(* CODESYS project ExampleRandomNumber.project

Project tree, tasks and I/O mapping:
  Device : CODESYS Control Win V3, 3S - Smart Software Solutions GmbH, order no. 305021, version 3.5.5.20
    application Application
      libraries: Standard, * (System)
      task MainTask (cyclic, interval t#20ms, priority 1) calls PLC_PRG_LD, PLC_PRG
      program PLC_PRG [ST]
      function rand [ST]
      global variables GVL
      program PLC_PRG_LD [LD]
  Rand/
    function rand [ST]
    program TestRand [ST]
*)

// Device/Application/GVL
VAR_GLOBAL
	randNext : ULINT := 42; //required external variable with a seed
END_VAR

// Device/Application/PLC_PRG_LD
//Test rand(), random number generator
PROGRAM PLC_PRG_LD
VAR
	number : UINT;
END_VAR

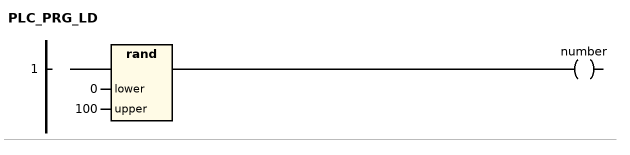
// NETWORK 1
number := rand(lower := 0, upper := 100);

END_PROGRAM

// Rand/rand
///Exempel: Generera slumptal mellan 1 ooch 10. 
///randNext : ULINT := 42;
///x : uint := rand(1,10)
///Ger ett slumptal mellan lower och upper
///Kräver att man har definierat en variabel randNext:ULINT:=<ett frö>;
///Ref: Bilting, U. Vägen Till C. Studentlitteratur. 2011.
FUNCTION rand : UINT
VAR_INPUT
	lower: UINT;
	upper: UINT;
END_VAR
VAR
	range: UINT := ((upper - lower) + 1);
	interval: UINT := (c4 / range);
	preRand: UINT;
END_VAR
VAR CONSTANT
	c1: UDINT := 1103515245;
	c2: UINT := 12345;
	c3: UDINT := 65536;
	c4: UINT := 32768;
END_VAR

randNext := randNext * c1 + c2;
preRand := ULINT_TO_UINT((randNext/c3) MOD c4);
IF interval > 0 THEN
	rand := (preRand+lower*interval-1)/interval; 
ELSE
	rand := preRand;
END_IF;
RETURN;

END_FUNCTION

// Device/Application/rand
//Example: Generate random numbers 1..10. 
//randNext : ULINT := 42; //required external variable with a seed
//x : uint := rand(1,10)
//
//Brief: Will give you a random number between lower och upper
//Requires an external variable: randNext:ULINT:=<seed>;
//Ref: Bilting, U. Vägen Till C. Studentlitteratur. 2011.
//
// Created by: Alexander Jaworowski 2015-02-05
// github.com/alexjaw/randomGenerator
FUNCTION rand : UINT
VAR_INPUT
	lower:UINT;
	upper:UINT;
END_VAR
VAR
	range:UINT:=upper-lower+1;
	interval:UINT:=c4/range;
	preRand:UINT;
END_VAR
VAR CONSTANT
	c1:UDINT:=1103515245;
	c2:UINT:=12345;
	c3:UDINT:=65536;
	c4:UINT:=32768;
END_VAR

randNext := randNext * c1 + c2;
preRand := ULINT_TO_UINT((randNext/c3) MOD c4);
IF interval > 0 THEN
	rand := (preRand+lower*interval-1)/interval; 
ELSE
	rand := preRand;
END_IF;
RETURN;

END_FUNCTION

// Device/Application/PLC_PRG
//Test rand(), random number generator
PROGRAM PLC_PRG
VAR
	number : UINT;
END_VAR

number := rand(lower:=0,upper:=42);

END_PROGRAM

// Rand/TestRand
PROGRAM TestRand
VAR
	randNext: ULINT := 42;
	x: UINT;
END_VAR

x := rand(1,10);

END_PROGRAM
